// TIA Portal V20 export
TYPE "SR-X100W_Read_Data"
   STRUCT
      "sr-x_100_Read_Data_1" : Char;
      "sr-x_100_Read_Data_2" : Char;
      "sr-x_100_Read_Data_3" : Char;
      "sr-x_100_Read_Data_4" : Char;
      "sr-x_100_Read_Data_5" : Char;
      "sr-x_100_Read_Data_6" : Char;
      "sr-x_100_Read_Data_7" : Char;
      "sr-x_100_Read_Data_8" : Char;
      "sr-x_100_Read_Data_9" : Char;
      "sr-x_100_Read_Data_10" : Char;
      "sr-x_100_Read_Data_11" : Char;
      "sr-x_100_Read_Data_12" : Char;
      "sr-x_100_Read_Data_13" : Char;
      "sr-x_100_Read_Data_14" : Char;
      "sr-x_100_Read_Data_15" : Char;
      "sr-x_100_Read_Data_16" : Char;
      "sr-x_100_Read_Data_17" : Char;
      "sr-x_100_Read_Data_18" : Char;
      "sr-x_100_Read_Data_19" : Char;
      "sr-x_100_Read_Data_20" : Char;
      "sr-x_100_Read_Data_21" : Char;
      "sr-x_100_Read_Data_22" : Char;
      "sr-x_100_Read_Data_23" : Char;
      "sr-x_100_Read_Data_24" : Char;
      "sr-x_100_Read_Data_25" : Char;
      "sr-x_100_Read_Data_26" : Char;
      "sr-x_100_Read_Data_27" : Char;
      "sr-x_100_Read_Data_28" : Char;
      "sr-x_100_Read_Data_29" : Char;
      "sr-x_100_Read_Data_30" : Char;
      "sr-x_100_Read_Data_31" : Char;
      "sr-x_100_Read_Data_32" : Char;
      "sr-x_100_Read_Data_33" : Char;
      "sr-x_100_Read_Data_34" : Char;
      "sr-x_100_Read_Data_35" : Char;
      "sr-x_100_Read_Data_36" : Char;
      "sr-x_100_Read_Data_37" : Char;
      "sr-x_100_Read_Data_38" : Char;
      "sr-x_100_Read_Data_39" : Char;
      "sr-x_100_Read_Data_40" : Char;
      "sr-x_100_Read_Data_41" : Char;
      "sr-x_100_Read_Data_42" : Char;
      "sr-x_100_Read_Data_43" : Char;
      "sr-x_100_Read_Data_44" : Char;
      "sr-x_100_Read_Data_45" : Char;
      "sr-x_100_Read_Data_46" : Char;
      "sr-x_100_Read_Data_47" : Char;
      "sr-x_100_Read_Data_48" : Char;
      "sr-x_100_Read_Data_49" : Char;
      "sr-x_100_Read_Data_50" : Char;
      "sr-x_100_Read_Data_51" : Char;
      "sr-x_100_Read_Data_52" : Char;
      "sr-x_100_Read_Data_53" : Char;
      "sr-x_100_Read_Data_54" : Char;
      "sr-x_100_Read_Data_55" : Char;
      "sr-x_100_Read_Data_56" : Char;
      "sr-x_100_Read_Data_57" : Char;
      "sr-x_100_Read_Data_58" : Char;
      "sr-x_100_Read_Data_59" : Char;
      "sr-x_100_Read_Data_60" : Char;
      "sr-x_100_Read_Data_61" : Char;
      "sr-x_100_Read_Data_62" : Char;
      "sr-x_100_Read_Data_63" : Char;
      "sr-x_100_Read_Data_64" : Char;
      "sr-x_100_Read_Data_65" : Char;
      "sr-x_100_Read_Data_66" : Char;
      "sr-x_100_Read_Data_67" : Char;
      "sr-x_100_Read_Data_68" : Char;
      "sr-x_100_Read_Data_69" : Char;
      "sr-x_100_Read_Data_70" : Char;
      "sr-x_100_Read_Data_71" : Char;
      "sr-x_100_Read_Data_72" : Char;
      "sr-x_100_Read_Data_73" : Char;
      "sr-x_100_Read_Data_74" : Char;
      "sr-x_100_Read_Data_75" : Char;
      "sr-x_100_Read_Data_76" : Char;
      "sr-x_100_Read_Data_77" : Char;
      "sr-x_100_Read_Data_78" : Char;
      "sr-x_100_Read_Data_79" : Char;
      "sr-x_100_Read_Data_80" : Char;
      "sr-x_100_Read_Data_81" : Char;
      "sr-x_100_Read_Data_82" : Char;
      "sr-x_100_Read_Data_83" : Char;
      "sr-x_100_Read_Data_84" : Char;
      "sr-x_100_Read_Data_85" : Char;
      "sr-x_100_Read_Data_86" : Char;
      "sr-x_100_Read_Data_87" : Char;
      "sr-x_100_Read_Data_88" : Char;
      "sr-x_100_Read_Data_89" : Char;
      "sr-x_100_Read_Data_90" : Char;
      "sr-x_100_Read_Data_91" : Char;
      "sr-x_100_Read_Data_92" : Char;
      "sr-x_100_Read_Data_93" : Char;
      "sr-x_100_Read_Data_94" : Char;
      "sr-x_100_Read_Data_95" : Char;
      "sr-x_100_Read_Data_96" : Char;
      "sr-x_100_Read_Data_97" : Char;
      "sr-x_100_Read_Data_98" : Char;
      "sr-x_100_Read_Data_99" : Char;
      "sr-x_100_Read_Data_100" : Char;
      "sr-x_100_Read_Data_101" : Char;
      "sr-x_100_Read_Data_102" : Char;
      "sr-x_100_Read_Data_103" : Char;
      "sr-x_100_Read_Data_104" : Char;
      "sr-x_100_Read_Data_105" : Char;
      "sr-x_100_Read_Data_106" : Char;
      "sr-x_100_Read_Data_107" : Char;
      "sr-x_100_Read_Data_108" : Char;
      "sr-x_100_Read_Data_109" : Char;
      "sr-x_100_Read_Data_110" : Char;
      "sr-x_100_Read_Data_111" : Char;
      "sr-x_100_Read_Data_112" : Char;
      "sr-x_100_Read_Data_113" : Char;
      "sr-x_100_Read_Data_114" : Char;
      "sr-x_100_Read_Data_115" : Char;
      "sr-x_100_Read_Data_116" : Char;
      "sr-x_100_Read_Data_117" : Char;
      "sr-x_100_Read_Data_118" : Char;
      "sr-x_100_Read_Data_119" : Char;
      "sr-x_100_Read_Data_120" : Char;
      "sr-x_100_Read_Data_121" : Char;
      "sr-x_100_Read_Data_122" : Char;
      "sr-x_100_Read_Data_123" : Char;
      "sr-x_100_Read_Data_124" : Char;
      "sr-x_100_Read_Data_125" : Char;
      "sr-x_100_Read_Data_126" : Char;
      "sr-x_100_Read_Data_127" : Char;
      "sr-x_100_Read_Data_128" : Char;
      "sr-x_100_Read_Data_129" : Char;
      "sr-x_100_Read_Data_130" : Char;
      "sr-x_100_Read_Data_131" : Char;
      "sr-x_100_Read_Data_132" : Char;
      "sr-x_100_Read_Data_133" : Char;
      "sr-x_100_Read_Data_134" : Char;
      "sr-x_100_Read_Data_135" : Char;
      "sr-x_100_Read_Data_136" : Char;
   END_STRUCT;
END_TYPE
